FUNCTION_BLOCK FB_MachineConfigure EXTENDS FB_Base IMPLEMENTS ITF_MachineConfigure
VAR
	(*	Baza konfiguracji	*)
	arritfConfigure				: ARRAY [0..10] OF ITF_Configuration;
	iNubmerOfAddedConfigure		: INT := -1;
END_VAR

METHOD PUBLIC AddConfiguration : BOOL
VAR_INPUT
	fbConfigure		: ITF_Configuration;
END_VAR
IF (THIS^.iNubmerOfAddedConfigure + 1 <= 10) THEN
	THIS^.iNubmerOfAddedConfigure	:= THIS^.iNubmerOfAddedConfigure + 1;
	THIS^.arritfConfigure [THIS^.iNubmerOfAddedConfigure]	:= fbConfigure;
	AddConfiguration	:= TRUE;
ELSE
	AddConfiguration	:= FALSE;
END_IF
END_METHOD

METHOD PUBLIC Configure : BOOL
VAR_INPUT
	fbMachineControl	: ITF_MachineControlConfigure;
END_VAR

VAR
	bResult				: BOOL;
	iI					: INT;
END_VAR
bResult			:= TRUE;

FOR iI := 0 TO THIS^.iNubmerOfAddedConfigure DO 
	IF (THIS^.arritfConfigure [iI] <> 0) THEN
		THIS^.arritfConfigure [iI].AddTopElementToMachineControl (itfMachineControl	:= fbMachineControl);
		THIS^.arritfConfigure [iI].AddTopElementToLogger ();
		THIS^.arritfConfigure [iI].StateAndModes (itfMachineControl := fbMachineControl);
		THIS^.arritfConfigure [iI].SetStartMode (itfMachineControl := fbMachineControl);
	END_IF
END_FOR

Configure		:= bResult;
END_METHOD

END_FUNCTION_BLOCK

(* stored: Version 1.1.0.1
   POU FB_MachineConfigure: Id {acdf548e-a6e8-4a73-8e7d-d1245eb04ae9}, SpecialFunc None
   Method AddConfiguration: Id {d9c2fdfe-2f2f-4e46-b4ba-30ce811a56ac}
   Method Configure: Id {f50fab32-d524-456f-8450-39a322865b3f} *)
